{attribute 'linkalways'} 
{attribute 'no_explicit_call' := 'This FB is a CLASS and must be accessed using methods or properties'}
{attribute 'enable_dynamic_creation'}
FUNCTION_BLOCK ParameterHost IMPLEMENTS I_Parameters, I_Serializable
VAR
	hostParent : I_HostParameters;
	eventTarget : I_EventTarget;
	parameters : Dictionary;
	selfCreatedParameters : Stack;
END_VAR

METHOD PUBLIC Accept
VAR_INPUT
	Visitor : I_ParameterVisitor;
END_VAR
VAR
	enumerator : I_ForwardEnumerator;
	parameter : I_Parameter;
END_VAR
enumerator := parameters.GetEnumerator();

WHILE (enumerator.MoveNext()) DO
	
	IF enumerator.TryGet(parameter) THEN
		parameter.Accept(Visitor);
	END_IF

END_WHILE

enumerator.Dispose();
END_METHOD

METHOD PUBLIC AddDataAsParameter : I_Parameter
VAR_INPUT
	Name : T_MAXSTRING;
	Data : I_Datatype;
END_VAR
VAR
	parameter : I_Parameter;
END_VAR
parameter := CreateParameter(Name, Data);
selfCreatedParameters.Push(parameter);
AddDataAsParameter := parameter;
END_METHOD

METHOD PUBLIC AddParameter
VAR_INPUT
	Parameter : I_Parameter;
END_VAR
parameters.AddOrUpdate(Parameter.Name, Parameter);
EmitOnParameterAddedEvent(Parameter);
END_METHOD

METHOD PRIVATE CreateParameter : I_Parameter
VAR_INPUT
	ParameterName : T_MAXSTRING;
	ParameterData : I_Datatype;
END_VAR
VAR
	pParameter : POINTER TO Parameter;
END_VAR
pParameter := __NEW(Parameter(Name := ParameterName, Data := ParameterData, Parent := hostParent));
CreateParameter := pParameter^;
END_METHOD

METHOD PRIVATE DisposeSelfCreatedParameters : BOOL
VAR
	parameter : I_Parameter;
END_VAR
WHILE selfCreatedParameters.TryPop(parameter) DO
	parameter.Dispose();
END_WHILE
END_METHOD

METHOD PROTECTED EmitOnParameterAddedEvent
VAR_INPUT
	Parameter : I_Parameter;
END_VAR
VAR
	pParameterAddedEvent : POINTER TO ParameterAddedEvent;
END_VAR
IF eventTarget = 0 THEN
	RETURN;
END_IF

pParameterAddedEvent := __NEW(ParameterAddedEvent(TargetParameter := Parameter));
eventTarget.Emit('OnParameterAdded',pParameterAddedEvent^);
pParameterAddedEvent^.Dispose();
END_METHOD

METHOD FB_exit : BOOL
VAR_INPUT
	bInCopyCode : BOOL; // if TRUE, the exit method is called for exiting an instance that is copied afterwards (online change).
END_VAR
IF bInCopyCode THEN
	RETURN;
END_IF

DisposeSelfCreatedParameters();
END_METHOD

METHOD FB_init : BOOL
VAR_INPUT
	bInitRetains : BOOL; // if TRUE, the retain variables are initialized (warm start / cold start)
	bInCopyCode : BOOL;  // if TRUE, the instance afterwards gets moved into the copy code (online change)
	Parent : I_HostParameters;
	ParentEventTarget : I_EventTarget;
END_VAR
hostParent := Parent;
eventTarget := ParentEventTarget;
END_METHOD

METHOD PUBLIC SerializeWith
VAR_INPUT
	Serializer : I_Serializer;
END_VAR
VAR
	enumerator : I_ForwardEnumerator;
	parameter : I_Parameter;
END_VAR
IF parameters.Count = 0 THEN
	RETURN;
END_IF

Serializer.AddKey('parameters');
Serializer.StartArray();

enumerator := parameters.GetEnumerator();

WHILE enumerator.MoveNext() DO
	IF enumerator.TryGet(parameter) THEN
		parameter.SerializeWith(Serializer);
	END_IF
END_WHILE

enumerator.Dispose();

Serializer.EndArray();
END_METHOD

METHOD PUBLIC TryDeserializeFrom : BOOL
VAR_INPUT
	Deserializer : I_Deserializer;
	Feedback : I_DeserializerFeedback;
END_VAR
VAR
	parametersDeserializer : I_Deserializer;
	parametersEnumerator : I_DeserializerObjectForwardEnumerator;
	parameter : I_Parameter;
END_VAR
parametersDeserializer := Deserializer.GetKeyObject('properties');
parametersEnumerator := parametersDeserializer.GetObjectEnumerator();

WHILE parametersEnumerator.MoveNext() DO
	
	IF NOT TryGetParameterByName(parametersEnumerator.Key, parameter) THEN
		CONTINUE;
	END_IF
	
	IF NOT parameter.TryDeserializeFrom(parametersEnumerator.Current, Feedback) THEN
		RETURN;
	END_IF

END_WHILE

parametersEnumerator.Dispose();
TryDeserializeFrom := TRUE;
END_METHOD

METHOD PUBLIC TryGetParameterByName : BOOL
VAR_INPUT
	Name : T_MAXSTRING;
	Destination : REFERENCE TO I_Parameter;
END_VAR
VAR
	parameter : I_Parameter;
END_VAR
IF NOT parameters.TryGetValue(Name, parameter) THEN
	RETURN;
END_IF

Destination := parameter;
TryGetParameterByName := TRUE;
END_METHOD

END_FUNCTION_BLOCK

(* stored: Version 1.1.0.1, ProductVersion 3.1.4024.12
   POU ParameterHost: Id {6bfffedc-4830-48d6-a087-df5e0f37d1bd}, SpecialFunc None
   Folder Constructor: Id {d962da93-42f3-408c-9e94-0c5674d47b60}
   Folder Destructor: Id {3738ba85-f78b-4784-bc7e-ba717d45d1fd}
   Folder Private: Id {579ccdeb-bdd6-417d-b99a-5960c5bca8fa}
   Folder Protected: Id {fa8eb0b0-8e53-404f-9aa4-b19cb7b4447d}
   Method Accept: Id {67a986cb-c3c8-4714-95da-82654735a15b}
   Method AddDataAsParameter: Id {170def95-49b8-459a-a221-caabe1bca48d}
   Method AddParameter: Id {62100911-1991-410b-b3b5-a2e6486a3099}
   Method CreateParameter: Id {6acdf74d-d8ae-4856-aa30-abaac77d646e}
   Method DisposeSelfCreatedParameters: Id {7784aab7-6df6-4fb6-bd06-2552ff15024a}
   Method EmitOnParameterAddedEvent: Id {2bfcadd9-8f8c-414b-8ace-7e1444c758d9}
   Method FB_exit: Id {13029f4e-91b6-4faa-833b-698cd56b2c4d}
   Method FB_init: Id {163161dd-2b78-474f-b1ea-d4408046e436}
   Method SerializeWith: Id {3efcd39e-7699-4bc3-a13e-91d6be2edb8c}
   Method TryDeserializeFrom: Id {68598c49-0246-4a15-9061-effd05f51e98}
   Method TryGetParameterByName: Id {ab07ca82-19c6-40f6-a546-6746aad8fa7f} *)
